// TwinCAT 3 PLC project DependencyInjectionPractice
// ProgramVersion: 3.1.4024.0
// libraries:
//   Tc2_Standard, * (Beckhoff Automation GmbH)
//   Tc2_System, * (Beckhoff Automation GmbH)
//   Tc3_Module, * (Beckhoff Automation GmbH)
// project tree:
//   / PlcTask.TcTTO
//   POUs/ FB_ConsoleLogger.TcPOU, FB_FileLogger.TcPOU, FB_Machine.TcPOU, I_Logger.TcIO, MAIN.TcPOU
// (motion and I/O tree: see PLC project functionblockpractice)
// real-time tasks:
//   TASK PlcTask: cycle T#10ms, priority 20, ADS port 350
//   TASK PlcTask2: cycle T#10ms, priority 22, ADS port 352
//   TASK PlcTask1: cycle T#10ms, priority 21, ADS port 351

CONFIGURATION DependencyInjectionPractice
    RESOURCE PLC ON TwinCAT3
        TASK PlcTask(INTERVAL := T#10ms, PRIORITY := 21);
        PROGRAM MAIN WITH PlcTask : MAIN;
    END_RESOURCE
END_CONFIGURATION

// ---- POUs/I_Logger.TcIO
INTERFACE I_Logger

METHOD M_Log : BOOL
VAR_INPUT
	sMessage : STRING(255);
END_VAR
END_METHOD

END_INTERFACE

// ---- POUs/MAIN.TcPOU
PROGRAM MAIN
VAR
	fbConsole1 : FB_ConsoleLogger;
	fbFile1 : FB_FileLogger;
	fbMachine1 : FB_Machine(fbFile1);
	fbMachine2 : FB_Machine(fbConsole1);
	
	sMessageStr1 : STRING(255):= 'This is printed in console ';
	sMessageStr2 : STRING(255) := 'This is written in file';
	
	bPass : BOOL := TRUE;
END_VAR

IF bPass THEN
	fbMachine1.M_Run(sMessageStr1);
	fbMachine2.M_Run(sMessageStr2);
	bPass := FALSE;
END_IF

END_PROGRAM

// ---- POUs/FB_ConsoleLogger.TcPOU
FUNCTION_BLOCK FB_ConsoleLogger IMPLEMENTS  I_Logger

VAR
END_VAR

{warning 'add method implementation '}
METHOD M_Log : BOOL
VAR_INPUT
	sMessage	: STRING(255);
END_VAR

ADSLOGSTR(msgCtrlMask:= ADSLOG_MSGTYPE_ERROR,
			msgFmtStr := 'Console log: %s',
			strArg := sMessage);
END_METHOD

END_FUNCTION_BLOCK

// ---- POUs/FB_FileLogger.TcPOU
FUNCTION_BLOCK FB_FileLogger IMPLEMENTS  I_Logger
VAR
END_VAR

{warning 'add method implementation '}
METHOD M_Log : BOOL
VAR_INPUT
	sMessage	: STRING(255);
END_VAR
ADSLOGSTR(
			msgCtrlMask:= ADSLOG_MSGTYPE_ERROR,
			msgFmtStr := 'File Log: %s',
			strArg := sMessage );
END_METHOD

END_FUNCTION_BLOCK

// ---- POUs/FB_Machine.TcPOU
FUNCTION_BLOCK FB_Machine

VAR
	iLogger : I_Logger;
END_VAR

METHOD FB_init : BOOL
VAR_INPUT
	bInitRetains : BOOL; // if TRUE, the retain variables are initialized (warm start / cold start)
	bInCopyCode : BOOL;  // if TRUE, the instance afterwards gets moved into the copy code (online change)
	_iLogger : I_Logger;
END_VAR
iLogger := _iLogger;
END_METHOD

METHOD M_Run : BOOL
VAR_INPUT
	sMessage : STRING(255);
END_VAR

IF iLogger <> 0 THEN
	iLogger.M_Log(sMessage);
END_IF
END_METHOD

END_FUNCTION_BLOCK
